FUNCTION_BLOCK E_TON (* standard timer function block (on-delay timing) *)
  (* Standard: 61499-2; Classification: standard timer function block; Description: Copyright (c) 2024 HR Agrartechnik GmbH This program and the accompanying materials are made available under the terms of the Eclipse Public License 2.0 which is available at https://www.eclipse.org/legal/epl-2.0/ SPDX-License-Identifier: EPL-2.0 *)
  (* Version 1.0, 2024-03-04, Franz Hoepfinger, HR Agrartechnik GmbH *)
  (* Version 3.0, 2025-04-14, Patrick Aigner, changed package *)
  PACKAGE iec61499::events::timers;
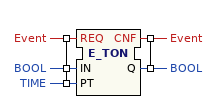
  EVENT_INPUT
    REQ WITH IN, PT; (* Normal Execution Request *)
  END_EVENT
  EVENT_OUTPUT
    CNF WITH Q; (* Execution Confirmation *)
  END_EVENT
  VAR_INPUT
    IN : BOOL; (* Input *)
    PT : TIME; (* Process time *)
  END_VAR
  VAR_OUTPUT
    Q : BOOL; (* Output *)
  END_VAR
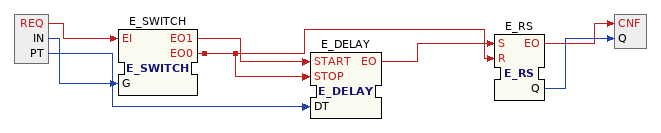
  FBS
    E_SWITCH : iec61499::events::E_SWITCH;
    E_DELAY : iec61499::events::E_DELAY;
    E_RS : iec61499::events::E_RS;
  END_FBS
  EVENT_CONNECTIONS
    REQ TO E_SWITCH.EI;
    E_SWITCH.EO1 TO E_DELAY.START;
    E_SWITCH.EO0 TO E_DELAY.STOP;
    E_DELAY.EO TO E_RS.S;
    E_SWITCH.EO0 TO E_RS.R;
    E_RS.EO TO CNF;
  END_CONNECTIONS
  DATA_CONNECTIONS
    IN TO E_SWITCH.G;
    PT TO E_DELAY.DT;
    E_RS.Q TO Q;
  END_CONNECTIONS
END_FUNCTION_BLOCK
